TYPE UA_OptionSet_Sample EXTENDS UA_OptionSet :
STRUCT
	BitOne : UA_OptionSet_Option;
	BitTwo : UA_OptionSet_Option;
END_STRUCT
END_TYPE

(* stored: Version 1.1.0.1
   DUT UA_OptionSet_Sample: Id {daa3661e-71ca-49b9-84ec-95c906721762} *)
